// TIA Portal V20 export
TYPE "LER_typeInventoryUDT"
// stored: Access Published
   STRUCT
      Input : Struct
         execute : Bool;
         attribute : Byte := 16#81;
         duration : Word := 16#1;
         durUnit : Word := 16#2;
      END_STRUCT;
      Output : Struct
         numberTags : Int;
         lengthData : Word;
         done : Bool;
         busy : Bool;
         error : Bool;
         status : DWord;
         pressence : Bool;
      END_STRUCT;
      InOut : Struct
         rfidData : Array[0..500] of Byte;
      END_STRUCT;
   END_STRUCT;
END_TYPE
